// TIA Portal V17 export
// export: Created 2024-06-16T17:47:24.9578887Z, ExportSetting WithDefaults, DisplayName Totally Integrated Automation Portal, DisplayVersion V17, DisplayName TIA Portal Openness, DisplayVersion V17, DisplayName TIA Portal Version Control Interface, DisplayVersion V17, DisplayName STEP 7 Professional, DisplayVersion V17, DisplayName STEP 7 Safety, DisplayVersion V17, DisplayName WinCC Professional, DisplayVersion V17
DATA_BLOCK "St1_In"   // DB105
{ S7_Optimized_Access := 'TRUE' }
VERSION : 0.1
// stored: AutoNumber false, DBAccessibleFromOPCUA true, DBAccessibleFromWebserver true, IsOnlyStoredInLoadMemory false, IsRetainMemResEnabled false, IsWriteProtectedInAS false, MemoryReserve 100
   VAR
      Pinces_Ouvert : Bool;   // Pinces de préhension Z : Ouverte
      Pinces_Fermee : Bool;   // Pinces de préhension Z : Fermée
      Cpt_C1 : Bool;   // Présence pile devant capteur Chargement AR : C1
      Cpt_C2 : Bool;   // Présence pile devant capteur Chargement AR : C2
      Cpt_C3 : Bool;   // Présence pile devant capteur Chargement AV : C3
      Cpt_C4 : Bool;   // Présence pile devant capteur Chargement AV : C4
      Cpt_C5 : Bool;   // Présence pile devant capteur Dépilement : C5
      Cpt_C6 : Bool;   // Détection collage barquette Dépilement : C6
      Cpt_C7 : Bool;   // Détection collage barquette Dépilement : C7
   END_VAR
BEGIN
END_DATA_BLOCK
